# EPICS autosave request: iocBoot/iocTomoScanStream_32ID/auto_settings.req
file "tomoScan_settings.req", P=$(P), R=$(R)
file "tomoScan_PSO_settings.req", P=$(P), R=$(R)
file "tomoScan_32ID_settings.req", P=$(P), R=$(R)
file "tomoScanStream_settings.req", P=$(P), R=$(R)
